(* IEC 61131-3 sources: dynamic-reversal/src/Blocks, 2 files *)

(* ---- LDR_CalcMoveAbsolute.st ---- *)
USING Siemens.S7.MotionControl;
USING System.Conversion;
USING System.FastMath;
NAMESPACE Simatic.Ax.LDR
    ///================================================================================
    /// SIEMENS AG
    /// (c)Copyright 2026 All Rights Reserved
    ///--------------------------------------------------------------------------------
    /// Library:       LDR
    /// Tested with:   FW 4.1
    /// Engineering:   SIMATIC AX
    /// Restrictions:  Should be called before the MC_MoveAbsolute block
    /// Requirements:  S7-1500
    /// Functionality: Calculation of interface signals for MC_MoveAbsolute to achieve
    ///                a dynamic reversal move without v=a=0
    ///================================================================================
    FUNCTION_BLOCK CalcMoveAbsolute
        VAR_INPUT
            /// Interconnect the axis here
            axis : DB_ANY;
            /// Rising edge: Starts the calculation of the Dynamic Reversal Move
            execute : BOOL;
            /// [Unit of TO] See MC_MoveAbsolute
            position : LREAL;
            /// [Unit of TO] See MC_MoveAbsolute
            velocity : LREAL := -1.0;
            /// [Unit of TO] See MC_MoveAbsolute
            acceleration : LREAL := -1.0;
            /// [Unit of TO] See MC_MoveAbsolute
            deceleration : LREAL := -1.0;
            /// [Unit of TO] See MC_MoveAbsolute
            jerk : LREAL := -1.0;
            /// [Unit of TO] See MC_MoveAbsolute. 1=Positive, 2=Negative, 3=Shortest
            direction : INT := 1;
            /// Interconnect the Output of the MC_Command.Busy here
            mcOutputBusy : BOOL;
            /// Interconnect the Output of the MC_Command.CommandAborted here
            mcOutputCommandAborted : BOOL;
            /// Interconnect the Output of the MC_Command.Error here
            mcOutputError : BOOL;
        END_VAR

        {S7.Extern := 'ReadOnly'}
        VAR_OUTPUT
            /// TRUE: Motion command reversed and command generation completed
            done : BOOL;
            /// TRUE: Function block active - motion calculation in progress
            busy : BOOL;
            /// TRUE: An error occurred during the execution of the FB
            error : BOOL;
            /// Further status information
            status : WORD := Status#NO_CALL;
            /// Connected to MC_MoveAbsolute.Execute input parameter
            mcExecute : BOOL;
            /// Connected to MC_MoveAbsolute.Position input parameter
            mcPosition : LREAL;
            /// Connected to MC_MoveAbsolute.Velocity input parameter
            mcVelocity : LREAL := -1.0;
            /// Connected to MC_MoveAbsolute.Acceleration input parameter
            mcAcceleration : LREAL := -1.0;
            /// Connected to MC_MoveAbsolute.Deceleration input parameter
            mcDeceleration : LREAL := -1.0;
            /// Connected to MC_MoveAbsolute.Jerk input parameter
            mcJerk : LREAL := -1.0;
            /// Connected to MC_MoveAbsolute.Direction input parameter
            mcDirection : INT := 1;
        END_VAR

        VAR
            _internal : typeInternal;
            _mainStateOld : FbState := FbState#NO_PROCESSING;
            _mainState : FbState := FbState#NO_PROCESSING;
            _mainStateEntry : BOOL;
            _positiveToNegativeTransition : BOOL;
            _negativeToPositiveTransition : BOOL;
            _dynamicProfilePossibleToBringZeroToTargetV : BOOL;
            _dynamicProfilePossibleToBringVToZero : BOOL;
            _aMaxStandardAfterZero : LREAL;
            _aMaxStandardBeforeZero : LREAL;
            _effectiveMcTargetJerk : LREAL;
            _effectiveMcTargetDeceleration : LREAL;
            _effectiveMcTargetAcceleration : LREAL;
            _effectiveMcTargetVelocity : LREAL;
            _initialToTargetDistance : LREAL;
            _absoluteDistanceToTarget : LREAL;
            _deltaPosition : LREAL;
            _distanceToBringVToZeroDynamic : LREAL;
            _distanceToBringVToZero : LREAL;
            _distanceAccelFromZeroDynamic : LREAL;
            _distanceAccelFromZero : LREAL;
            _minDistanceAfterZeroCross : LREAL;
            _totalRequiredDistanceDynamic : LREAL;
            _totalRequiredDistance : LREAL;
            _jerkTime : LREAL;
            _accelReachedVelocity : LREAL;
        END_VAR

        VAR_TEMP
            tempExecute : BOOL;
            tempAxisStartupData : typeAxisStartupData;
            tempAxisCyclicData : typeAxisCyclicData;
        END_VAR

        VAR CONSTANT
            PRECISION_FACTOR : LREAL := 100.0;
        END_VAR

        // --- TRIGGERING ---
        tempExecute := execute;
        IF (tempExecute = TRUE) AND (_internal.executePrevious = FALSE)
            AND (_internal.output.status = Status#NO_CALL)
        THEN
            // --- INIT ---
            _internal.output.done := FALSE;
            _internal.output.busy := TRUE;
            _internal.output.error := FALSE;
            _internal.output.mcExecute := FALSE;
            _internal.output.mcPosition := 0.0;
            _internal.output.mcVelocity := 0.0;
            _internal.output.mcAcceleration := 0.0;
            _internal.output.mcDeceleration := 0.0;
            _internal.output.mcJerk := 0.0;

            tempAxisStartupData := GetTOStartupData(axis := axis);
            _internal.input.toModuloEnabled := tempAxisStartupData.toModuloEnabled;
            _internal.input.toModuloLength := tempAxisStartupData.toModuloLength;
            _internal.input.toModuloStartvalue := tempAxisStartupData.toModuloStartvalue;
            _internal.input.toDefaultVelocity := tempAxisStartupData.toDefaultVelocity;
            _internal.input.toDefaultAcceleration := tempAxisStartupData.toDefaultAcceleration;
            _internal.input.toDefaultDeceleration := tempAxisStartupData.toDefaultDeceleration;
            _internal.input.toDefaultJerk := tempAxisStartupData.toDefaultJerk;
            _internal.input.toMaxVelocity := tempAxisStartupData.toMaxVelocity;
            _internal.input.toMaxAcceleration := tempAxisStartupData.toMaxAcceleration;
            _internal.input.toMaxDeceleration := tempAxisStartupData.toMaxDeceleration;
            _internal.input.toMaxJerk := tempAxisStartupData.toMaxJerk;
            _internal.input.toPosition := tempAxisStartupData.toPosition;
            _internal.input.toVelocity := tempAxisStartupData.toVelocity;
            _internal.input.mcTargetPosition := position;
            _internal.input.mcTargetVelocity := velocity;
            _internal.input.mcTargetAcceleration := acceleration;
            _internal.input.mcTargetDeceleration := deceleration;
            _internal.input.mcTargetJerk := jerk;
            _internal.input.mcTargetDirection := direction;
            _internal.input.typeOfTO := tempAxisStartupData.typeOfTO;
            _initialToTargetDistance := _internal.input.mcTargetPosition - _internal.input.toPosition;
            _absoluteDistanceToTarget := 0.0;
            _deltaPosition := 0.0;
            _distanceToBringVToZero := 0.0;
            _distanceAccelFromZero := 0.0;
            _minDistanceAfterZeroCross := 0.0;
            _totalRequiredDistance := 0.0;
            _jerkTime := 0.0;
            _accelReachedVelocity := 0.0;
            _dynamicProfilePossibleToBringVToZero := FALSE;
            _dynamicProfilePossibleToBringZeroToTargetV := FALSE;

            // --- CHECK INVALID INPUT ---
            //TO check - must be positioning axis at least
            IF _internal.input.typeOfTO <= 1 THEN
                _internal.output.status := Errors#AXIS_TYPE;
            END_IF;

            //Position check - target position must be within the modulo range
            IF _internal.input.toModuloEnabled AND
                (_internal.input.mcTargetPosition < _internal.input.toModuloStartvalue
                OR _internal.input.mcTargetPosition > (_internal.input.toModuloStartvalue + _internal.input.toModuloLength))
            THEN
                _internal.output.status := Errors#POSITION_OUT_OF_MODULO_BOUNDARY;
            END_IF;

            //Velocity check
            IF _internal.input.mcTargetVelocity >= _internal.input.toMaxVelocity THEN
                IF (_internal.output.status AND WORD#16#8000) <> WORD#16#8000 THEN
                    _internal.output.status := Warnings#MC_TARGET_VELOCITY_EXCEEDS_MAX;
                END_IF;
                _internal.input.mcTargetVelocity := _internal.input.toMaxVelocity;
                _effectiveMcTargetVelocity := _internal.input.mcTargetVelocity;
            ELSIF _internal.input.mcTargetVelocity = 0.0 THEN
                _internal.output.status := Errors#MC_INVALID_ZERO_DYNAMICS;
            ELSIF _internal.input.mcTargetVelocity < 0.0 THEN
                _effectiveMcTargetVelocity := _internal.input.toDefaultVelocity;
            ELSE
                _effectiveMcTargetVelocity := _internal.input.mcTargetVelocity;
            END_IF;

            //Acceleration check
            IF _internal.input.mcTargetAcceleration >= _internal.input.toMaxAcceleration THEN
                IF (_internal.output.status AND WORD#16#8000) <> WORD#16#8000 THEN
                    _internal.output.status := Warnings#MC_TARGET_ACCELERATION_EXCEEDS_MAX;
                END_IF;
                _internal.input.mcTargetAcceleration := _internal.input.toMaxAcceleration;
                _effectiveMcTargetAcceleration := _internal.input.toMaxAcceleration;
            ELSIF _internal.input.mcTargetAcceleration = 0.0 THEN
                _internal.output.status := Errors#MC_INVALID_ZERO_DYNAMICS;
            ELSIF _internal.input.mcTargetAcceleration < 0.0 THEN
                _effectiveMcTargetAcceleration := _internal.input.toDefaultAcceleration;
            ELSE
                _effectiveMcTargetAcceleration := _internal.input.mcTargetAcceleration;
            END_IF;

            //Deceleration check
            IF _internal.input.mcTargetDeceleration >= _internal.input.toMaxDeceleration THEN
                IF (_internal.output.status AND WORD#16#8000) <> WORD#16#8000 THEN
                    _internal.output.status := Warnings#MC_TARGET_DECELERATION_EXCEEDS_MAX;
                END_IF;
                _internal.input.mcTargetDeceleration := _internal.input.toMaxDeceleration;
                _effectiveMcTargetDeceleration := _internal.input.toMaxDeceleration;
            ELSIF _internal.input.mcTargetDeceleration = 0.0 THEN
                _internal.output.status := Errors#MC_INVALID_ZERO_DYNAMICS;
            ELSIF _internal.input.mcTargetDeceleration < 0.0 THEN
                _effectiveMcTargetDeceleration := _internal.input.toDefaultDeceleration;
            ELSE
                _effectiveMcTargetDeceleration := _internal.input.mcTargetDeceleration;
            END_IF;

            //Jerk check
            IF _internal.input.mcTargetJerk >= _internal.input.toMaxJerk THEN
                IF (_internal.input.mcTargetJerk = 0.0) OR (_internal.input.toMaxJerk = 0.0) THEN
                    _internal.input.mcTargetJerk := 0.0;
                    _effectiveMcTargetJerk := 1.0e+12;
                ELSE
                    IF (_internal.output.status AND WORD#16#8000) <> WORD#16#8000 THEN
                        _internal.output.status := Warnings#MC_TARGET_JERK_EXCEEDS_MAX;
                    END_IF;
                    _internal.input.mcTargetJerk := _internal.input.toMaxJerk;
                END_IF;
            ELSIF _internal.input.mcTargetJerk < 0.0 THEN
                _effectiveMcTargetJerk := _internal.input.toDefaultJerk;
            ELSE
                _effectiveMcTargetJerk := _internal.input.mcTargetJerk;
            END_IF;

            //Direction check
            IF (_internal.input.mcTargetDirection = 1) AND _internal.input.toModuloEnabled THEN
                _effectiveMcTargetVelocity := _effectiveMcTargetVelocity * 1.0;
            ELSIF (_internal.input.mcTargetDirection = 2) AND _internal.input.toModuloEnabled THEN
                _effectiveMcTargetVelocity := _effectiveMcTargetVelocity * -1.0;
            ELSIF (_internal.input.mcTargetDirection = 3) OR NOT _internal.input.toModuloEnabled THEN
                IF NOT _internal.input.toModuloEnabled THEN
                    IF _internal.input.toPosition > _internal.input.mcTargetPosition THEN
                        _effectiveMcTargetVelocity := _effectiveMcTargetVelocity * -1.0;
                    ELSE
                        _effectiveMcTargetVelocity := _effectiveMcTargetVelocity * 1.0;
                    END_IF;
                ELSE
                    IF (_initialToTargetDistance >= 0.0) AND (ABS(_initialToTargetDistance) <= 0.5 * _internal.input.toModuloLength) THEN
                        _effectiveMcTargetVelocity := _effectiveMcTargetVelocity * 1.0;
                    ELSIF (_initialToTargetDistance < 0.0) AND (ABS(_initialToTargetDistance) <= 0.5 * _internal.input.toModuloLength) THEN
                        _effectiveMcTargetVelocity := _effectiveMcTargetVelocity * -1.0;
                    ELSIF (_initialToTargetDistance >= 0.0) AND (ABS(_initialToTargetDistance) > 0.5 * _internal.input.toModuloLength) THEN
                        _effectiveMcTargetVelocity := _effectiveMcTargetVelocity * -1.0;
                    ELSE
                        _effectiveMcTargetVelocity := _effectiveMcTargetVelocity * 1.0;
                    END_IF;
                END_IF;
            ELSE
                _internal.output.status := Errors#MC_DIRECTION_INVALID;
            END_IF;

            IF _internal.output.status = Status#NO_CALL THEN
                _internal.output.status := Status#FIRST_CALL;
            END_IF;

            _positiveToNegativeTransition := (_internal.input.toVelocity > 0)
                                             AND (_effectiveMcTargetVelocity < 0)
                                             AND (_internal.input.mcTargetJerk <> 0);
            _negativeToPositiveTransition := (_internal.input.toVelocity < 0)
                                             AND (_effectiveMcTargetVelocity > 0)
                                             AND (_internal.input.mcTargetJerk <> 0);

            // --- FEASIBILITY CHECK ---
            IF (_internal.input.toModuloEnabled AND (_internal.input.mcTargetDirection = 3))
                OR NOT _internal.input.toModuloEnabled
            THEN
                _deltaPosition := _internal.input.mcTargetPosition - _internal.input.toPosition;
                IF _deltaPosition > (_internal.input.toModuloLength / 2.0) THEN
                    _deltaPosition := _deltaPosition - _internal.input.toModuloLength;
                ELSIF _deltaPosition < (- _internal.input.toModuloLength / 2.0) THEN
                    _deltaPosition := _deltaPosition + _internal.input.toModuloLength;
                END_IF;
                _absoluteDistanceToTarget := ABS(_deltaPosition);
            ELSE
                _absoluteDistanceToTarget := ABS(_initialToTargetDistance);
            END_IF;

            IF (_positiveToNegativeTransition OR _negativeToPositiveTransition) AND (_effectiveMcTargetJerk > 0.0) THEN
                //Distance to bring velocity to zero
                IF (ABS(_internal.input.toVelocity) > 0.0) AND (_effectiveMcTargetDeceleration > 0.0) THEN
                    _jerkTime := _effectiveMcTargetDeceleration / _effectiveMcTargetJerk;
                    _accelReachedVelocity := 0.5 * _effectiveMcTargetJerk * _jerkTime * _jerkTime;
                    IF ABS(_internal.input.toVelocity) <= _accelReachedVelocity THEN
                        _distanceToBringVToZero := (2.0 / 3.0) * ABS(_internal.input.toVelocity)
                                                   * SQRT(2.0 * ABS(_internal.input.toVelocity) / _effectiveMcTargetJerk);
                        _dynamicProfilePossibleToBringVToZero := FALSE;
                    ELSE
                        _distanceToBringVToZero := (ABS(_internal.input.toVelocity) * ABS(_internal.input.toVelocity)
                                                   / (2.0 * _effectiveMcTargetDeceleration)) + (_effectiveMcTargetDeceleration
                                                   * ABS(_internal.input.toVelocity) / (2.0 * _effectiveMcTargetJerk));
                        _distanceToBringVToZeroDynamic := _distanceToBringVToZero / 2.0;
                        _dynamicProfilePossibleToBringVToZero := TRUE;
                    END_IF;
                ELSE
                    _distanceToBringVToZero := 0.0;
                END_IF;

                //Distance to accelerate from zero to target velocity
                IF (ABS(_effectiveMcTargetVelocity) > 0.0) AND (_effectiveMcTargetAcceleration > 0.0)
                    AND (_effectiveMcTargetDeceleration > 0.0)
                THEN
                    _jerkTime := _effectiveMcTargetAcceleration / _effectiveMcTargetJerk;
                    _accelReachedVelocity := 0.5 * _effectiveMcTargetJerk * _jerkTime * _jerkTime;
                    IF ABS(_effectiveMcTargetVelocity) <= _accelReachedVelocity THEN
                        _distanceAccelFromZero := (2.0 / 3.0) * ABS(_effectiveMcTargetVelocity) * SQRT(2.0 * ABS(_effectiveMcTargetVelocity) / _effectiveMcTargetJerk);
                        _dynamicProfilePossibleToBringZeroToTargetV := FALSE;
                    ELSE
                        _distanceAccelFromZero := (ABS(_effectiveMcTargetVelocity) * ABS(_effectiveMcTargetVelocity) / (2.0 * _effectiveMcTargetAcceleration)) + (_effectiveMcTargetAcceleration * ABS(_effectiveMcTargetVelocity) / (2.0 * _effectiveMcTargetJerk));
                        _distanceAccelFromZeroDynamic := _distanceAccelFromZero / 2.0;
                        _dynamicProfilePossibleToBringZeroToTargetV := TRUE;
                    END_IF;
                ELSE
                    _distanceAccelFromZero := 0.0;
                END_IF;

                _totalRequiredDistance := _distanceToBringVToZero + _distanceAccelFromZero;
                _totalRequiredDistanceDynamic := _distanceToBringVToZeroDynamic + _distanceAccelFromZeroDynamic;

                IF NOT _dynamicProfilePossibleToBringZeroToTargetV OR NOT _dynamicProfilePossibleToBringVToZero
                    OR (_totalRequiredDistanceDynamic >= _absoluteDistanceToTarget)
                THEN
                    IF _internal.output.status < WORD#16#7500 THEN
                        _internal.output.status := Warnings#NO_DYNAMIC_REVERSAL_POSSIBLE;
                    END_IF;
                END_IF;
            END_IF;

            // --- INIT STATE SELECTION ---
            IF (_internal.output.status AND WORD#16#8000) = WORD#16#8000 THEN
                _mainState := FbState#NO_PROCESSING;
            ELSIF _internal.output.status = Warnings#NO_DYNAMIC_REVERSAL_POSSIBLE THEN
                _mainState := FbState#PROCESSING_THIRD_JERK_LIMITATION;
            ELSIF (_positiveToNegativeTransition OR _negativeToPositiveTransition) THEN
                _mainState := FbState#PROCESSING_FIRST_JERK_LIMITATION;
            ELSE
                IF _effectiveMcTargetJerk = 0.0 THEN
                    _internal.output.status := Warnings#NO_DYNAMIC_REVERSAL_NEEDED_TRAPEZOID_CHOSEN;
                ELSE
                    _internal.output.status := Warnings#NO_REVERSAL_NEEDED;
                END_IF;
                _mainState := FbState#PROCESSING_THIRD_JERK_LIMITATION;
            END_IF;
        ELSIF (_internal.output.status = Status#FIRST_CALL) THEN
            _internal.output.status := Status#SUBSEQUENT_CALL;
        END_IF;
        _internal.executePrevious := tempExecute;

        // --- CYCLIC ---
        IF (_internal.output.status = Status#NO_CALL) THEN
            RETURN;
        END_IF;
        IF (_internal.output.status > Status#NO_CALL) AND (_internal.output.status < Status#GENERAL_ERROR) THEN
            tempAxisCyclicData := GetTOCyclicData(axis := axis, requestPosition := FALSE);
            _internal.input.toVelocity := tempAxisCyclicData.toVelocity;
            _internal.input.toAcceleration := tempAxisCyclicData.toAcceleration;
            _internal.input.mcOutputBusy := mcOutputBusy;
            _internal.input.mcOutputError := mcOutputError;
            _internal.input.mcOutputCommandAborted := mcOutputCommandAborted;
            IF _internal.input.mcOutputCommandAborted THEN
                _internal.output.status := Errors#MC_COMMAND_ABORTED;
                _mainState := FbState#NO_PROCESSING;
            END_IF;
            IF _mainStateOld <> _mainState THEN
                _mainStateEntry := TRUE;
            ELSE
                _mainStateEntry := FALSE;
            END_IF;
            _mainStateOld := _mainState;
        END_IF;

        // --- STATE MACHINE ---
        CASE _mainState OF
            FbState#NO_PROCESSING:
                ;

            FbState#PROCESSING_FIRST_JERK_LIMITATION:
                _internal.output.mcPosition := _internal.input.mcTargetPosition;
                _internal.output.mcDirection := _internal.input.mcTargetDirection;
                _internal.output.mcVelocity := _internal.input.mcTargetVelocity;
                _internal.output.mcAcceleration := _internal.input.mcTargetAcceleration;
                _internal.output.mcDeceleration := _internal.input.mcTargetDeceleration;
                _internal.output.mcJerk := _internal.input.mcTargetJerk;
                _internal.output.mcExecute := TRUE;

                IF _internal.input.mcOutputError THEN
                    _internal.output.mcExecute := FALSE;
                    _internal.output.status := Errors#MC_COMMAND_IN_ERROR;
                END_IF;

                IF _internal.input.mcOutputBusy
                    AND _internal.output.mcExecute
                    AND NOT _mainStateEntry
                THEN
                    _mainState := FbState#PROCESSING_SECOND_CROSSING_ZERO_VELOCITY;
                END_IF;

            FbState#PROCESSING_SECOND_CROSSING_ZERO_VELOCITY:
                IF (_positiveToNegativeTransition AND (_internal.input.toVelocity <= 0))
                    OR (_negativeToPositiveTransition AND (_internal.input.toVelocity >= 0))
                THEN
                    _mainState := FbState#PROCESSING_THIRD_JERK_LIMITATION;
                    RETURN;
                END_IF;

                IF _mainStateEntry THEN
                    _internal.output.mcExecute := FALSE;
                ELSE
                    IF _positiveToNegativeTransition THEN
                        IF ROUND(_internal.input.toAcceleration * PRECISION_FACTOR) = ROUND(- _effectiveMcTargetDeceleration * PRECISION_FACTOR)
                        THEN
                            _internal.output.mcPosition := _internal.input.mcTargetPosition;
                            _internal.output.mcDirection := _internal.input.mcTargetDirection;
                            _internal.output.mcVelocity := _internal.input.mcTargetVelocity;
                            _internal.output.mcAcceleration := _internal.input.mcTargetAcceleration;
                            _internal.output.mcDeceleration := _internal.input.mcTargetDeceleration;
                            _internal.output.mcJerk := 0.0;
                            _internal.output.mcExecute := TRUE;
                        END_IF;
                    ELSIF _negativeToPositiveTransition THEN
                        IF ROUND(_internal.input.toAcceleration * PRECISION_FACTOR) = ROUND(_effectiveMcTargetAcceleration * PRECISION_FACTOR)
                        THEN
                            _internal.output.mcPosition := _internal.input.mcTargetPosition;
                            _internal.output.mcDirection := _internal.input.mcTargetDirection;
                            _internal.output.mcVelocity := _internal.input.mcTargetVelocity;
                            _internal.output.mcAcceleration := _internal.input.mcTargetAcceleration;
                            _internal.output.mcDeceleration := _internal.input.mcTargetDeceleration;
                            _internal.output.mcJerk := 0.0;
                            _internal.output.mcExecute := TRUE;
                        END_IF;
                    END_IF;
                END_IF;

                IF _internal.input.mcOutputError THEN
                    _internal.output.mcExecute := FALSE;
                    _internal.output.status := Errors#MC_COMMAND_IN_ERROR;
                END_IF;

                IF _internal.input.mcOutputBusy
                    AND _internal.output.mcExecute
                    AND NOT _mainStateEntry
                THEN
                    _mainState := FbState#PROCESSING_THIRD_JERK_LIMITATION;
                END_IF;

            FbState#PROCESSING_THIRD_JERK_LIMITATION:
                IF _mainStateEntry
                    AND NOT (_internal.output.status = Warnings#NO_REVERSAL_NEEDED)
                    AND NOT (_internal.output.status = Warnings#NO_DYNAMIC_REVERSAL_POSSIBLE)
                    AND NOT (_internal.output.status = Warnings#NO_DYNAMIC_REVERSAL_NEEDED_TRAPEZOID_CHOSEN)
                THEN
                    _internal.output.mcExecute := FALSE;
                ELSE
                    IF (_positiveToNegativeTransition AND (_internal.input.toVelocity < 0)) OR
                        (_negativeToPositiveTransition AND (_internal.input.toVelocity > 0)) OR
                        (_internal.output.status = Warnings#NO_REVERSAL_NEEDED) OR
                        (_internal.output.status = Warnings#NO_DYNAMIC_REVERSAL_POSSIBLE) OR
                        (_internal.output.status = Warnings#NO_DYNAMIC_REVERSAL_NEEDED_TRAPEZOID_CHOSEN)
                    THEN
                        _internal.output.mcPosition := _internal.input.mcTargetPosition;
                        _internal.output.mcDirection := _internal.input.mcTargetDirection;
                        _internal.output.mcVelocity := _internal.input.mcTargetVelocity;
                        _internal.output.mcAcceleration := _internal.input.mcTargetAcceleration;
                        _internal.output.mcDeceleration := _internal.input.mcTargetDeceleration;
                        _internal.output.mcJerk := _internal.input.mcTargetJerk;
                        _internal.output.mcExecute := TRUE;
                    END_IF;

                    IF _internal.input.mcOutputError THEN
                        _internal.output.mcExecute := FALSE;
                        _internal.output.status := Errors#MC_COMMAND_IN_ERROR;
                    END_IF;

                    IF _internal.input.mcOutputBusy
                        AND _internal.output.mcExecute
                        AND NOT _mainStateEntry
                    THEN
                        _internal.output.status := Status#EXECUTION_FINISHED;
                    END_IF;
                END_IF;
            ELSE
                ; //Unexpected state
        END_CASE;

        // --- OUTPUTS ---
        IF (_internal.output.status = Status#EXECUTION_FINISHED) AND (_internal.output.done = FALSE) THEN
            _internal.output.done := TRUE;
            _internal.output.busy := FALSE;
            _internal.output.error := FALSE;
            _mainState := FbState#NO_PROCESSING;
        ELSIF ((_internal.output.status AND WORD#16#8000) = WORD#16#8000) AND (_internal.output.error = FALSE) THEN
            _internal.output.done := FALSE;
            _internal.output.busy := FALSE;
            _internal.output.error := TRUE;
            _mainState := FbState#NO_PROCESSING;
        ELSIF (tempExecute = FALSE) AND ((_internal.output.done = TRUE) OR (_internal.output.error = TRUE)) THEN
            _internal.output.done := FALSE;
            _internal.output.busy := FALSE;
            _internal.output.error := FALSE;
            _internal.output.status := Status#NO_CALL;
            _internal.output.mcExecute := FALSE;
            _internal.output.mcPosition := 0.0;
            _internal.output.mcDirection := 1;
            _internal.output.mcVelocity := -1.0;
            _internal.output.mcAcceleration := -1.0;
            _internal.output.mcDeceleration := -1.0;
            _internal.output.mcJerk := -1.0;
        END_IF;

        done := _internal.output.done;
        busy := _internal.output.busy;
        error := _internal.output.error;
        status := _internal.output.status;
        mcExecute := _internal.output.mcExecute;
        mcPosition := _internal.output.mcPosition;
        mcDirection := _internal.output.mcDirection;
        mcVelocity := _internal.output.mcVelocity;
        mcAcceleration := _internal.output.mcAcceleration;
        mcDeceleration := _internal.output.mcDeceleration;
        mcJerk := _internal.output.mcJerk;
    END_FUNCTION_BLOCK
END_NAMESPACE

(* ---- LDR_CalcMoveVelocity.st ---- *)
USING Siemens.S7.MotionControl;
USING System.Conversion;
USING System.FastMath;
NAMESPACE Simatic.Ax.LDR
    ///================================================================================
    /// SIEMENS AG
    /// (c)Copyright 2026 All Rights Reserved
    ///--------------------------------------------------------------------------------
    /// Library:       LDR
    /// Tested with:   FW 4.1
    /// Engineering:   SIMATIC AX
    /// Restrictions:  Should be called before the MC_MoveVelocity block
    /// Requirements:  S7-1500
    /// Functionality: Calculation of interface signals for MC_MoveVelocity to achieve
    ///                a dynamic reversal move without v=a=0
    ///================================================================================
    FUNCTION_BLOCK CalcMoveVelocity
        VAR_INPUT
            /// Interconnect the axis here
            axis : DB_ANY;
            /// Rising edge: Starts the calculation of the Dynamic Reversal Move
            execute : BOOL;
            /// [Unit of TO] See MC_MoveVelocity. Can be 0.0 (unlike MC_MoveAbsolute)
            velocity : LREAL := 100.0;
            /// [Unit of TO] See MC_MoveVelocity
            acceleration : LREAL := -1.0;
            /// [Unit of TO] See MC_MoveVelocity
            deceleration : LREAL := -1.0;
            /// [Unit of TO] See MC_MoveVelocity
            jerk : LREAL := -1.0;
            /// [Unit of TO] See MC_MoveVelocity. 0=Use sign of Velocity, 1=Positive, 2=Negative
            direction : INT;
            /// Interconnect the Output of the MC_Command.Busy here
            mcOutputBusy : BOOL;
            /// Interconnect the Output of the MC_Command.CommandAborted here
            mcOutputCommandAborted : BOOL;
            /// Interconnect the Output of the MC_Command.Error here
            mcOutputError : BOOL;
        END_VAR

        {S7.Extern := 'ReadOnly'}
        VAR_OUTPUT
            /// TRUE: Motion command reversed and final command generation completed
            done : BOOL;
            /// TRUE: Function block active - motion calculation in progress
            busy : BOOL;
            /// TRUE: An error occurred during the execution of the FB
            error : BOOL;
            /// Further status information
            status : WORD := Status#NO_CALL;
            /// Connected to MC_MoveVelocity.Execute input parameter
            mcExecute : BOOL;
            /// Connected to MC_MoveVelocity.Velocity input parameter
            mcVelocity : LREAL := -1.0;
            /// Connected to MC_MoveVelocity.Acceleration input parameter
            mcAcceleration : LREAL := -1.0;
            /// Connected to MC_MoveVelocity.Deceleration input parameter
            mcDeceleration : LREAL := -1.0;
            /// Connected to MC_MoveVelocity.Jerk input parameter
            mcJerk : LREAL := -1.0;
            /// Connected to MC_MoveVelocity.Direction input parameter
            mcDirection : INT;
        END_VAR

        VAR
            _internal : typeInternal;
            _mainStateOld : FbState := FbState#NO_PROCESSING;
            _mainState : FbState := FbState#NO_PROCESSING;
            _mainStateEntry : BOOL;
            _positiveToNegativeTransition : BOOL;
            _negativeToPositiveTransition : BOOL;
            _dynamicProfilePossibleToBringZeroToTargetV : BOOL;
            _dynamicProfilePossibleToBringVToZero : BOOL;
            _effectiveMcTargetJerk : LREAL;
            _effectiveMcTargetDeceleration : LREAL;
            _effectiveMcTargetAcceleration : LREAL;
            _effectiveMcTargetVelocity : LREAL;
            _jerkTime : LREAL;
            _accelReachedVelocity : LREAL;
        END_VAR

        VAR_TEMP
            tempExecute : BOOL;
            tempAxisStartupData : typeAxisStartupData;
            tempAxisCyclicData : typeAxisCyclicData;
        END_VAR

        VAR CONSTANT
            PRECISION_FACTOR : LREAL := 100.0;
        END_VAR

        // --- TRIGGERING ---
        tempExecute := execute;
        IF (tempExecute = TRUE) AND (_internal.executePrevious = FALSE)
            AND (_internal.output.status = Status#NO_CALL)
        THEN
            // --- INIT ---
            _internal.output.done := FALSE;
            _internal.output.busy := TRUE;
            _internal.output.error := FALSE;
            _internal.output.mcExecute := FALSE;
            _internal.output.mcVelocity := 0.0;
            _internal.output.mcAcceleration := 0.0;
            _internal.output.mcDeceleration := 0.0;
            _internal.output.mcJerk := 0.0;
            _internal.output.mcDirection := 0;

            tempAxisStartupData := GetTOStartupData(axis := axis);
            _internal.input.toDefaultVelocity := tempAxisStartupData.toDefaultVelocity;
            _internal.input.toDefaultAcceleration := tempAxisStartupData.toDefaultAcceleration;
            _internal.input.toDefaultDeceleration := tempAxisStartupData.toDefaultDeceleration;
            _internal.input.toDefaultJerk := tempAxisStartupData.toDefaultJerk;
            _internal.input.toMaxVelocity := tempAxisStartupData.toMaxVelocity;
            _internal.input.toMaxAcceleration := tempAxisStartupData.toMaxAcceleration;
            _internal.input.toMaxDeceleration := tempAxisStartupData.toMaxDeceleration;
            _internal.input.toMaxJerk := tempAxisStartupData.toMaxJerk;
            _internal.input.toVelocity := tempAxisStartupData.toVelocity;
            _internal.input.mcTargetVelocity := velocity;
            _internal.input.mcTargetAcceleration := acceleration;
            _internal.input.mcTargetDeceleration := deceleration;
            _internal.input.mcTargetJerk := jerk;
            _internal.input.mcTargetDirection := direction;
            _internal.input.typeOfTO := tempAxisStartupData.typeOfTO;
            _jerkTime := 0.0;
            _accelReachedVelocity := 0.0;
            _dynamicProfilePossibleToBringVToZero := FALSE;
            _dynamicProfilePossibleToBringZeroToTargetV := FALSE;

            // --- CHECK INVALID INPUT ---
            IF _internal.input.typeOfTO < 1 THEN
                _internal.output.status := Errors#AXIS_TYPE;
            END_IF;

            //Velocity check - can be any value including 0.0 (MoveVelocity specific)
            IF ABS(_internal.input.mcTargetVelocity) >= _internal.input.toMaxVelocity THEN
                IF (_internal.output.status AND WORD#16#8000) <> WORD#16#8000 THEN
                    _internal.output.status := Warnings#MC_TARGET_VELOCITY_EXCEEDS_MAX;
                END_IF;
                IF _internal.input.mcTargetVelocity >= 0.0 THEN
                    _internal.input.mcTargetVelocity := _internal.input.toMaxVelocity;
                ELSE
                    _internal.input.mcTargetVelocity := - _internal.input.toMaxVelocity;
                END_IF;
            END_IF;
            _effectiveMcTargetVelocity := _internal.input.mcTargetVelocity;

            //Acceleration check
            IF _internal.input.mcTargetAcceleration >= _internal.input.toMaxAcceleration THEN
                IF (_internal.output.status AND WORD#16#8000) <> WORD#16#8000 THEN
                    _internal.output.status := Warnings#MC_TARGET_ACCELERATION_EXCEEDS_MAX;
                END_IF;
                _internal.input.mcTargetAcceleration := _internal.input.toMaxAcceleration;
                _effectiveMcTargetAcceleration := _internal.input.toMaxAcceleration;
            ELSIF _internal.input.mcTargetAcceleration = 0.0 THEN
                _internal.output.status := Errors#MC_INVALID_ZERO_DYNAMICS;
            ELSIF _internal.input.mcTargetAcceleration < 0.0 THEN
                _effectiveMcTargetAcceleration := _internal.input.toDefaultAcceleration;
            ELSE
                _effectiveMcTargetAcceleration := _internal.input.mcTargetAcceleration;
            END_IF;

            //Deceleration check
            IF _internal.input.mcTargetDeceleration >= _internal.input.toMaxDeceleration THEN
                IF (_internal.output.status AND WORD#16#8000) <> WORD#16#8000 THEN
                    _internal.output.status := Warnings#MC_TARGET_DECELERATION_EXCEEDS_MAX;
                END_IF;
                _internal.input.mcTargetDeceleration := _internal.input.toMaxDeceleration;
                _effectiveMcTargetDeceleration := _internal.input.toMaxDeceleration;
            ELSIF _internal.input.mcTargetDeceleration = 0.0 THEN
                _internal.output.status := Errors#MC_INVALID_ZERO_DYNAMICS;
            ELSIF _internal.input.mcTargetDeceleration < 0.0 THEN
                _effectiveMcTargetDeceleration := _internal.input.toDefaultDeceleration;
            ELSE
                _effectiveMcTargetDeceleration := _internal.input.mcTargetDeceleration;
            END_IF;

            //Jerk check
            IF _internal.input.mcTargetJerk >= _internal.input.toMaxJerk THEN
                IF (_internal.input.mcTargetJerk = 0.0) OR (_internal.input.toMaxJerk = 0.0) THEN
                    _internal.input.mcTargetJerk := 0.0;
                    _effectiveMcTargetJerk := 1.0e+12;
                ELSE
                    IF (_internal.output.status AND WORD#16#8000) <> WORD#16#8000 THEN
                        _internal.output.status := Warnings#MC_TARGET_JERK_EXCEEDS_MAX;
                    END_IF;
                    _internal.input.mcTargetJerk := _internal.input.toMaxJerk;
                END_IF;
            ELSIF _internal.input.mcTargetJerk < 0.0 THEN
                _effectiveMcTargetJerk := _internal.input.toDefaultJerk;
            ELSE
                _effectiveMcTargetJerk := _internal.input.mcTargetJerk;
            END_IF;

            //Direction check - MoveVelocity specific: 0, 1, 2 only
            IF _internal.input.mcTargetDirection = 0 THEN
                ;
            ELSIF _internal.input.mcTargetDirection = 1 THEN
                _effectiveMcTargetVelocity := ABS(_effectiveMcTargetVelocity);
            ELSIF _internal.input.mcTargetDirection = 2 THEN
                _effectiveMcTargetVelocity := - ABS(_effectiveMcTargetVelocity);
            ELSE
                _internal.output.status := Errors#MC_DIRECTION_INVALID;
            END_IF;

            IF _internal.output.status = Status#NO_CALL THEN
                _internal.output.status := Status#FIRST_CALL;
            END_IF;

            //Calculate transitions
            _positiveToNegativeTransition := (_internal.input.toVelocity > 0) AND (_effectiveMcTargetVelocity < 0) AND (_internal.input.mcTargetJerk <> 0);
            _negativeToPositiveTransition := (_internal.input.toVelocity < 0) AND (_effectiveMcTargetVelocity > 0) AND (_internal.input.mcTargetJerk <> 0);

            // --- CHECK DYNAMIC REVERSAL FEASIBILITY ---
            IF (_positiveToNegativeTransition OR _negativeToPositiveTransition) AND (_effectiveMcTargetJerk > 0.0) THEN
                //Deceleration phase check
                IF (ABS(_internal.input.toVelocity) > 0.0) AND (_effectiveMcTargetDeceleration > 0.0) THEN
                    _jerkTime := _effectiveMcTargetDeceleration / _effectiveMcTargetJerk;
                    _accelReachedVelocity := 0.5 * _effectiveMcTargetJerk * _jerkTime * _jerkTime;
                    IF ABS(_internal.input.toVelocity) <= _accelReachedVelocity THEN
                        _dynamicProfilePossibleToBringVToZero := FALSE;
                    ELSE
                        _dynamicProfilePossibleToBringVToZero := TRUE;
                    END_IF;
                ELSE
                    _dynamicProfilePossibleToBringVToZero := FALSE;
                END_IF;

                //Acceleration phase check
                IF (ABS(_effectiveMcTargetVelocity) > 0.0) AND (_effectiveMcTargetAcceleration > 0.0) THEN
                    _jerkTime := _effectiveMcTargetAcceleration / _effectiveMcTargetJerk;
                    _accelReachedVelocity := 0.5 * _effectiveMcTargetJerk * _jerkTime * _jerkTime;
                    IF ABS(_effectiveMcTargetVelocity) <= _accelReachedVelocity THEN
                        _dynamicProfilePossibleToBringZeroToTargetV := FALSE;
                    ELSE
                        _dynamicProfilePossibleToBringZeroToTargetV := TRUE;
                    END_IF;
                ELSE
                    _dynamicProfilePossibleToBringZeroToTargetV := FALSE;
                END_IF;

                IF NOT _dynamicProfilePossibleToBringZeroToTargetV OR NOT _dynamicProfilePossibleToBringVToZero THEN
                    IF _internal.output.status < WORD#16#7500 THEN
                        _internal.output.status := Warnings#NO_DYNAMIC_REVERSAL_POSSIBLE;
                    END_IF;
                END_IF;
            END_IF;

            // --- INIT STATE SELECTION ---
            IF (_internal.output.status AND WORD#16#8000) = WORD#16#8000 THEN
                _mainState := FbState#NO_PROCESSING;
            ELSIF _internal.output.status = Warnings#NO_DYNAMIC_REVERSAL_POSSIBLE THEN
                _mainState := FbState#PROCESSING_THIRD_JERK_LIMITATION;
            ELSIF (_positiveToNegativeTransition OR _negativeToPositiveTransition) THEN
                _mainState := FbState#PROCESSING_FIRST_JERK_LIMITATION;
            ELSE
                IF _effectiveMcTargetJerk = 0.0 THEN
                    _internal.output.status := Warnings#NO_DYNAMIC_REVERSAL_NEEDED_TRAPEZOID_CHOSEN;
                ELSE
                    _internal.output.status := Warnings#NO_REVERSAL_NEEDED;
                END_IF;
                _mainState := FbState#PROCESSING_THIRD_JERK_LIMITATION;
            END_IF;
        ELSIF (_internal.output.status = Status#FIRST_CALL) THEN
            _internal.output.status := Status#SUBSEQUENT_CALL;
        END_IF;
        _internal.executePrevious := tempExecute;

        // --- CYCLIC ---
        IF (_internal.output.status = Status#NO_CALL) THEN
            RETURN;
        END_IF;
        IF (_internal.output.status > Status#NO_CALL) AND (_internal.output.status < Status#GENERAL_ERROR) THEN
            tempAxisCyclicData := GetTOCyclicData(axis := axis, requestPosition := FALSE);
            _internal.input.toVelocity := tempAxisCyclicData.toVelocity;
            _internal.input.toAcceleration := tempAxisCyclicData.toAcceleration;
            _internal.input.mcOutputBusy := mcOutputBusy;
            _internal.input.mcOutputError := mcOutputError;
            _internal.input.mcOutputCommandAborted := mcOutputCommandAborted;
            IF _internal.input.mcOutputCommandAborted THEN
                _internal.output.status := Errors#MC_COMMAND_ABORTED;
                _mainState := FbState#NO_PROCESSING;
            END_IF;
            IF _mainStateOld <> _mainState THEN
                _mainStateEntry := TRUE;
            ELSE
                _mainStateEntry := FALSE;
            END_IF;
            _mainStateOld := _mainState;
        END_IF;

        // --- STATE MACHINE ---
        CASE _mainState OF
            FbState#NO_PROCESSING:
                ; //No processing active

            FbState#PROCESSING_FIRST_JERK_LIMITATION:
                _internal.output.mcDirection := _internal.input.mcTargetDirection;
                _internal.output.mcVelocity := _internal.input.mcTargetVelocity;
                _internal.output.mcAcceleration := _internal.input.mcTargetAcceleration;
                _internal.output.mcDeceleration := _internal.input.mcTargetDeceleration;
                _internal.output.mcJerk := _internal.input.mcTargetJerk;
                _internal.output.mcExecute := TRUE;

                IF _internal.input.mcOutputError THEN
                    _internal.output.mcExecute := FALSE;
                    _internal.output.status := Errors#MC_COMMAND_IN_ERROR;
                END_IF;

                IF _internal.input.mcOutputBusy
                    AND _internal.output.mcExecute
                    AND NOT _mainStateEntry
                THEN
                    _mainState := FbState#PROCESSING_SECOND_CROSSING_ZERO_VELOCITY;
                END_IF;

            FbState#PROCESSING_SECOND_CROSSING_ZERO_VELOCITY:
                //Check if already crossed zero
                IF (_positiveToNegativeTransition AND (_internal.input.toVelocity < 0))
                    OR (_negativeToPositiveTransition AND (_internal.input.toVelocity > 0))
                THEN
                    _mainState := FbState#PROCESSING_THIRD_JERK_LIMITATION;
                    RETURN;
                END_IF;

                IF _mainStateEntry THEN
                    _internal.output.mcExecute := FALSE;
                ELSE
                    IF _positiveToNegativeTransition THEN
                        IF ROUND(_internal.input.toAcceleration * PRECISION_FACTOR) = ROUND(- _effectiveMcTargetDeceleration * PRECISION_FACTOR)
                        THEN
                            _internal.output.mcDirection := _internal.input.mcTargetDirection;
                            _internal.output.mcVelocity := _internal.input.mcTargetVelocity;
                            _internal.output.mcAcceleration := _internal.input.mcTargetAcceleration;
                            _internal.output.mcDeceleration := _internal.input.mcTargetDeceleration;
                            _internal.output.mcJerk := 0.0;
                            _internal.output.mcExecute := TRUE;
                        END_IF;
                    ELSIF _negativeToPositiveTransition THEN
                        IF ROUND(_internal.input.toAcceleration * PRECISION_FACTOR) = ROUND(_effectiveMcTargetAcceleration * PRECISION_FACTOR)
                        THEN
                            _internal.output.mcDirection := _internal.input.mcTargetDirection;
                            _internal.output.mcVelocity := _internal.input.mcTargetVelocity;
                            _internal.output.mcAcceleration := _internal.input.mcTargetAcceleration;
                            _internal.output.mcDeceleration := _internal.input.mcTargetDeceleration;
                            _internal.output.mcJerk := 0.0;
                            _internal.output.mcExecute := TRUE;
                        END_IF;
                    END_IF;
                END_IF;

                IF _internal.input.mcOutputError THEN
                    _internal.output.mcExecute := FALSE;
                    _internal.output.status := Errors#MC_COMMAND_IN_ERROR;
                END_IF;

                IF _internal.input.mcOutputBusy
                    AND _internal.output.mcExecute
                    AND NOT _mainStateEntry
                THEN
                    _mainState := FbState#PROCESSING_THIRD_JERK_LIMITATION;
                END_IF;

            FbState#PROCESSING_THIRD_JERK_LIMITATION:
                IF _mainStateEntry
                    AND NOT (_internal.output.status = Warnings#NO_REVERSAL_NEEDED)
                    AND NOT (_internal.output.status = Warnings#NO_DYNAMIC_REVERSAL_POSSIBLE)
                    AND NOT (_internal.output.status = Warnings#NO_DYNAMIC_REVERSAL_NEEDED_TRAPEZOID_CHOSEN)
                THEN
                    _internal.output.mcExecute := FALSE;
                ELSE
                    IF (_positiveToNegativeTransition AND (_internal.input.toVelocity < 0)) OR
                        (_negativeToPositiveTransition AND (_internal.input.toVelocity > 0)) OR
                        (_internal.output.status = Warnings#NO_REVERSAL_NEEDED) OR
                        (_internal.output.status = Warnings#NO_DYNAMIC_REVERSAL_POSSIBLE) OR
                        (_internal.output.status = Warnings#NO_DYNAMIC_REVERSAL_NEEDED_TRAPEZOID_CHOSEN)
                    THEN
                        _internal.output.mcDirection := _internal.input.mcTargetDirection;
                        _internal.output.mcVelocity := _internal.input.mcTargetVelocity;
                        _internal.output.mcAcceleration := _internal.input.mcTargetAcceleration;
                        _internal.output.mcDeceleration := _internal.input.mcTargetDeceleration;
                        _internal.output.mcJerk := _internal.input.mcTargetJerk;
                        _internal.output.mcExecute := TRUE;
                    END_IF;

                    IF _internal.input.mcOutputError THEN
                        _internal.output.mcExecute := FALSE;
                        _internal.output.status := Errors#MC_COMMAND_IN_ERROR;
                    END_IF;

                    IF _internal.input.mcOutputBusy
                        AND _internal.output.mcExecute
                        AND NOT _mainStateEntry
                    THEN
                        _internal.output.status := Status#EXECUTION_FINISHED;
                    END_IF;
                END_IF;
            ELSE
                ; //Unexpected state
        END_CASE;

        // --- OUTPUTS ---
        IF (_internal.output.status = Status#EXECUTION_FINISHED) AND (_internal.output.done = FALSE) THEN
            _internal.output.done := TRUE;
            _internal.output.busy := FALSE;
            _internal.output.error := FALSE;
            _mainState := FbState#NO_PROCESSING;
        ELSIF ((_internal.output.status AND WORD#16#8000) = WORD#16#8000) AND (_internal.output.error = FALSE) THEN
            _internal.output.done := FALSE;
            _internal.output.busy := FALSE;
            _internal.output.error := TRUE;
            _mainState := FbState#NO_PROCESSING;
        ELSIF (tempExecute = FALSE) AND ((_internal.output.done = TRUE) OR (_internal.output.error = TRUE)) THEN
            _internal.output.done := FALSE;
            _internal.output.busy := FALSE;
            _internal.output.error := FALSE;
            _internal.output.status := Status#NO_CALL;
            _internal.output.mcExecute := FALSE;
            _internal.output.mcDirection := 0;
            _internal.output.mcVelocity := -1.0;
            _internal.output.mcAcceleration := -1.0;
            _internal.output.mcDeceleration := -1.0;
            _internal.output.mcJerk := -1.0;
        END_IF;

        done := _internal.output.done;
        busy := _internal.output.busy;
        error := _internal.output.error;
        status := _internal.output.status;
        mcExecute := _internal.output.mcExecute;
        mcDirection := _internal.output.mcDirection;
        mcVelocity := _internal.output.mcVelocity;
        mcAcceleration := _internal.output.mcAcceleration;
        mcDeceleration := _internal.output.mcDeceleration;
        mcJerk := _internal.output.mcJerk;
    END_FUNCTION_BLOCK
END_NAMESPACE
